// TIA Portal V16 export
// export: Created 2022-09-01T13:58:57.5606986Z, ExportSetting WithDefaults, DisplayName Totally Integrated Automation Portal, DisplayVersion V16, DisplayName TIA Portal Version Control Interface, DisplayVersion V16, DisplayName TIA Portal Openness, DisplayVersion V16, DisplayName STEP 7 Professional, DisplayVersion V16, DisplayName STEP 7 Safety, DisplayVersion V16, DisplayName WinCC Advanced, DisplayVersion V16
FUNCTION "T_Func_Bombas" : Void   // FC9, LAD
{ S7_Optimized_Access := 'TRUE' }
VERSION : 0.1
// stored: AutoNumber true, IsIECCheckEnabled false, SetENOAutomatically false, UDAEnableTagReadback false
   VAR_TEMP   // added for the SCL form of the ladder/FBD networks
      _w1 : Bool;
   END_VAR
BEGIN

REGION Network 1: Período de tempo de alternancia das bombas
   // Se contador = 0, trabalha B1 e B2. Se = 1, trabalha B1 e B3. Se = 2, trabalha B2 e B3
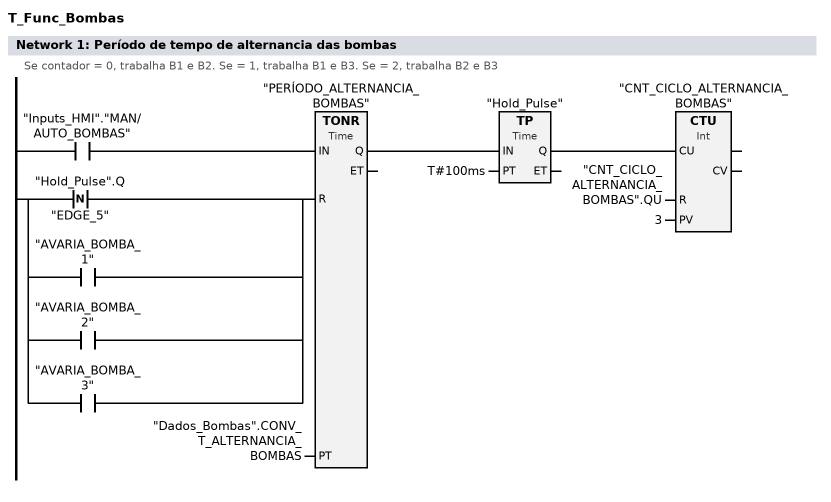
   RUNG wire#powerrail
      Contact( "Inputs_HMI"."MAN/AUTO_BOMBAS" )
      { S7_Templates := "time_type := Time" } "PERÍODO_ALTERNANCIA_BOMBAS".TONR(r := wire#w1, pt := "Dados_Bombas".CONV_T_ALTERNANCIA_BOMBAS, et =>)
      { S7_Templates := "time_type := Time" } "Hold_Pulse".TP(pt := T#100ms, et =>)
      { S7_Templates := "value_type := Int" } "CNT_CICLO_ALTERNANCIA_BOMBAS".CTU(r := "CNT_CICLO_ALTERNANCIA_BOMBAS".QU, pv := 3, cv =>)
   END_RUNG
   RUNG wire#powerrail
      N_Contact(operand := "Hold_Pulse".Q, bit := "EDGE_5")
   END_RUNG wire#w1
   RUNG wire#powerrail
      Contact( "AVARIA_BOMBA_1" )
   END_RUNG wire#w1
   RUNG wire#powerrail
      Contact( "AVARIA_BOMBA_2" )
   END_RUNG wire#w1
   RUNG wire#powerrail
      Contact( "AVARIA_BOMBA_3" )
   END_RUNG wire#w1
   // the same network as SCL:
   #_w1 := NOT "Hold_Pulse".Q AND "EDGE_5";   // falling edge of "Hold_Pulse".Q
   "EDGE_5" := "Hold_Pulse".Q;
   "PERÍODO_ALTERNANCIA_BOMBAS".TONR(IN := "Inputs_HMI"."MAN/AUTO_BOMBAS",
                           R := #_w1 OR "AVARIA_BOMBA_1" OR "AVARIA_BOMBA_2" OR "AVARIA_BOMBA_3",
                           PT := "Dados_Bombas".CONV_T_ALTERNANCIA_BOMBAS);
   "Hold_Pulse".TP(IN := "PERÍODO_ALTERNANCIA_BOMBAS".Q, PT := T#100ms);
   "CNT_CICLO_ALTERNANCIA_BOMBAS".CTU(CU := "Hold_Pulse".Q, R := "CNT_CICLO_ALTERNANCIA_BOMBAS".QU, PV := 3);
END_REGION
END_FUNCTION
